{attribute 'GeneratedUsingTerminal: EK1100-0000-0018'}
{attribute addProperty BoxType "EK1100-0000-0018"}
{attribute addProperty Id "Term_15_EL3403EL3403_200C424073Term_16_EK1122Term_16_EK1122_E3300954164Term_23_EL3024EL3024_C4269E3248"}
{attribute addProperty CRC "3983405165"}
{attribute addProperty Size "285"}
TYPE Term_14_EK1100_ED6DF06D EXTENDS EK1100_1FC0878B :
STRUCT
	{attribute addProperty Name "Term_15_EL3403"}
	{attribute addProperty PreviousPort "Term 14 (EK1100) : B"}
	Term_15_EL3403 : EL3403_200C4240;
	{attribute addProperty Name "Term_16_EK1122"}
	{attribute addProperty PreviousPort "Term 15 (EL3403) : B"}
	Term_16_EK1122 : Term_16_EK1122_E3300954;
	{attribute addProperty Name "Term_23_EL3024"}
	{attribute addProperty PreviousPort "Term 16 (EK1122) : C"}
	Term_23_EL3024 : EL3024_C4269E32;
END_STRUCT
END_TYPE

(* stored: Version 1.2.0.0, ProductVersion 3.1.4024.9
   DUT Term_14_EK1100_ED6DF06D: Id {366ce184-7503-069b-02c8-453c48cc86b3} *)
